FUNCTION_BLOCK PUBLIC OB_StopBeforeVisionStation
VAR_INPUT
END_VAR
VAR_OUTPUT
END_VAR
VAR
	xTrigger :BOOL := FALSE; // triggers processing
	State : eOB_StopBeforeVisionState := eOB_StopBeforeVisionState.eUnknown;
	NextState : eOB_StopBeforeVisionState := eOB_StopBeforeVisionState.eUnknown;
	bFirst : BOOL := TRUE;
	VUT : BYTE; //VehicleID Under Station
	DwellTimer : TON;
END_VAR

CASE State OF

eOB_StopBeforeVisionState.eUnknown:
	NextState := eOB_StopBeforeVisionState.eReady;

eOB_StopBeforeVisionState.eInit:

eOB_StopBeforeVisionState.eHoming:

eOB_StopBeforeVisionState.eReady:
	IF (xTrigger) THEN
		NextState := eOB_StopBeforeVisionState.eDwell;		
		DwellTimer(IN:=FALSE);
	END_IF

eOB_StopBeforeVisionState.eDwell:
	DwellTimer(IN:=TRUE, PT := T#600MS);
	IF (GVL_IO.VS_XPartPresentBeforeVision) THEN 
		PartsData.Status[VUT].OverallStatus := ePartStatus.eLoaded;
        NextState := eOB_StopBeforeVisionState.eProcessing;		
		DwellTimer(IN:=FALSE);
	END_IF
	IF (DwellTimer.Q) THEN // just call it loaded, no sensor is present 
		NextState := eOB_StopBeforeVisionState.eProcessing;		
		PartsData.Status[VUT].OverallStatus := ePartStatus.eLoaded;
		DwellTimer(IN:=FALSE);
	END_IF

eOB_StopBeforeVisionState.eProcessing:
	IF (NOT Stations.fbVisionSta.InspectionOnGoing) THEN
		NextState := eOB_StopBeforeVisionState.eDepart;
	END_IF

eOB_StopBeforeVisionState.eDepart:
	    UpdatePartData();
		Stations.fbRoutePlanner.M_NotifyVehStaCmpl(StationIndex:= MM_CONST.STOP_BEFORE_VISION_STA, VehicleID := VUT);
		xTrigger := FALSE;
		NextState := eOB_StopBeforeVisionState.eReady;

eOB_StopBeforeVisionState.eError:
END_CASE

IF (State <> NextState) THEN
	bFirst := TRUE;
ELSE
	bFirst := FALSE;
END_IF

State := NextState;

METHOD PUBLIC ClearVehicleTrigger : BOOL
VAR_INPUT
END_VAR
xTrigger := FALSE;
END_METHOD

PROPERTY PUBLIC Trigger : BOOL
SET
xTrigger := Trigger;
END_SET
END_PROPERTY

METHOD PUBLIC UpdatePartData : BOOL
VAR_INPUT
END_VAR
PartsData.Status[VUT].BurnOffTemp := GVL_IO.BU_Temperature/10;
END_METHOD

PROPERTY PUBLIC VehicleUnderTest : BYTE
GET
VehicleUnderTest := VUT;
END_GET
SET
VUT := VehicleUnderTest;
END_SET
END_PROPERTY

END_FUNCTION_BLOCK

(* stored: Version 1.1.0.1, ProductVersion 3.1.4022.6
   POU OB_StopBeforeVisionStation: Id {5cb07ee7-8d9e-4d49-bedd-4859912012a9}, SpecialFunc None
   Method ClearVehicleTrigger: Id {2e1c596d-5d2b-4639-b99e-5f6e5ea3a76c}
   Property Trigger: Id {ee49aa6e-a684-4efa-b494-49869a69f2a3}
   Set Set: Id {b26aa3a0-8028-4325-bea7-afd6d08367c3}
   Method UpdatePartData: Id {2d06d4a0-4e96-434d-96a9-4783573025fb}
   Property VehicleUnderTest: Id {267ec9f2-69c2-425c-8b48-3a21d0dfa33f}
   Get Get: Id {7bda8d34-9c37-4a52-87e5-0d6623766a7c}
   Set Set: Id {9ff98e18-9a4c-4722-af08-4027456e344c} *)
